FUNCTION_BLOCK ManStartFlushGSI (* Basic Function Block Type *)
  (* Standard: 61499-2 *)
  (* Version 0.0, 6/20/2026, Schneider Electric, Template *)
  PACKAGE SE.Nereda;
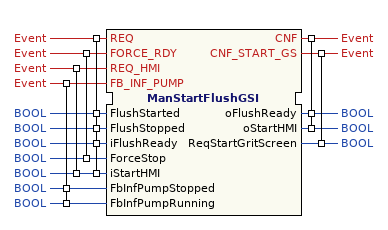
  EVENT_INPUT
    REQ WITH FlushStarted, FlushStopped, iFlushReady, iStartHMI; (* Normal Execution Request *)
    FORCE_RDY WITH ForceStop;
    REQ_HMI WITH iStartHMI;
    FB_INF_PUMP WITH FbInfPumpStopped, FbInfPumpRunning;
  END_EVENT
  EVENT_OUTPUT
    CNF WITH oFlushReady, oStartHMI; (* Execution Confirmation *)
    CNF_START_GS WITH ReqStartGritScreen;
  END_EVENT
  VAR_INPUT
    FlushStarted : BOOL;
    FlushStopped : BOOL;
    iFlushReady : BOOL;
    ForceStop : BOOL;
    iStartHMI : BOOL;
    FbInfPumpStopped : BOOL;
    FbInfPumpRunning : BOOL;
  END_VAR
  VAR_OUTPUT
    oFlushReady : BOOL;
    oStartHMI : BOOL;
    ReqStartGritScreen : BOOL;
  END_VAR
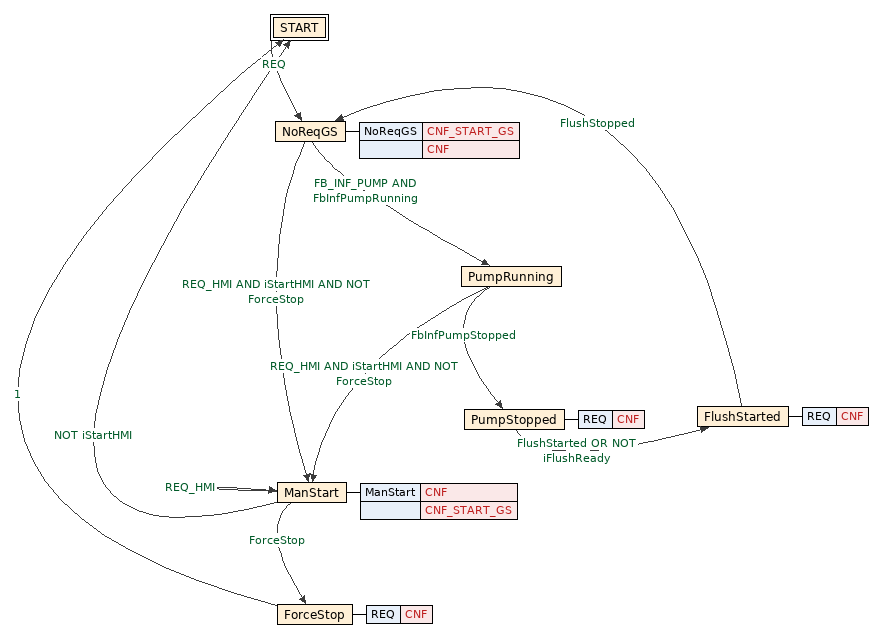
  EC_STATES
    START; (* Initial State *)
    PumpRunning;
    ManStart : ManStart -> CNF, -> CNF_START_GS;
    ForceStop : REQ -> CNF;
    NoReqGS : NoReqGS -> CNF_START_GS, -> CNF;
    PumpStopped : REQ -> CNF;
    FlushStarted : REQ -> CNF;
  END_STATES
  EC_TRANSITIONS
    START TO NoReqGS := REQ;
    NoReqGS TO ManStart := REQ_HMI AND iStartHMI AND NOT ForceStop;
    ManStart TO ManStart := REQ_HMI;
    ManStart TO START := NOT iStartHMI;
    ManStart TO ForceStop := ForceStop;
    ForceStop TO START := 1;
    NoReqGS TO PumpRunning := FB_INF_PUMP AND FbInfPumpRunning;
    PumpRunning TO PumpStopped := FbInfPumpStopped;
    PumpRunning TO ManStart := REQ_HMI AND iStartHMI AND NOT ForceStop;
    PumpStopped TO FlushStarted := FlushStarted OR NOT iFlushReady;
    FlushStarted TO NoReqGS := FlushStopped;
  END_TRANSITIONS
  ALGORITHM REQ IN ST:
;
oFlushReady := iFlushReady;
  END_ALGORITHM
  ALGORITHM ManStart IN ST:
;
oFlushReady := TRUE;
oStartHMI := iStartHMI;
ReqStartGritScreen := TRUE;
  END_ALGORITHM
  ALGORITHM NoReqGS IN ST:
;
ReqStartGritScreen := FALSE;
oFlushReady := FALSE;
  END_ALGORITHM
END_FUNCTION_BLOCK
